(* PLC project poST.project, poSTIDE *)
(* stored: creationDateTime 2021-08-31T00:00:00.000000 *)

FUNCTION DIVTIME : TIME
  VAR_INPUT
    in1 : TIME;
    in2 : ANY_NUM;
  END_VAR

END_FUNCTION
